{attribute 'GeneratedUsingTerminal: EK1100-0000-0018'}
{attribute addProperty BoxType "EK1100-0000-0018"}
{attribute addProperty Id "Beckhoff_ER5xxxEK1122Beckhoff_ER5xxxEK1122_B89AF081104"}
{attribute addProperty CRC "581225248"}
{attribute addProperty Size "104"}
TYPE Beckhoff_ER5xxx_22A4CB20 EXTENDS EK1100_1FC0878B :
STRUCT
	{attribute addProperty Name "Beckhoff_ER5xxxEK1122"}
	Beckhoff_ER5xxxEK1122 : Beckhoff_ER5xxxEK1122_B89AF081;
END_STRUCT
END_TYPE

(* stored: Version 1.2.0.0, ProductVersion 3.1.4024.9
   DUT Beckhoff_ER5xxx_22A4CB20: Id {029a65ed-18cd-4b93-ba43-03d8ea6e9304} *)
